INTERFACE I_EpicsMotionParamsStatus

METHOD MotionParamsAndStatus
VAR_INPUT
	PowerEnabled : BOOL;
	PowerIsEnabled : BOOL;
	Execute : BOOL;
	LimHome : BOOL;
	MoveBackwardEnabled : BOOL;
	MoveForwardEnabled : BOOL;
	MeasuredPositionDiff : LREAL;
	MeasuredPosition : LREAL;
	MeasuredVelocity : LREAL;
	PowerOverride : LREAL;
	Busy : BOOL;
	HomeDone : BOOL;
END_VAR
END_METHOD

END_INTERFACE

(* stored: Version 1.1.0.1
   Itf I_EpicsMotionParamsStatus: Id {bfb903e2-9136-49f8-be52-58ed07e3baa9}
   Method MotionParamsAndStatus: Id {b23cbd51-01d2-4f59-93b6-a0f074fb8271} *)
